TYPE T_FileExtension : STRING[4];
END_TYPE

(* stored: Version 1.1.0.1, ProductVersion 3.1.4024.15
   DUT T_FileExtension: Id {9506d373-93bb-4515-a2f0-36db9be22e12} *)
